{attribute 'qualified_only'}
{attribute 'strict'}
{attribute 'to_string'}
TYPE eTcaStorageCmd :
(
	noCmd := 0,
	FillCarrier,
	RemoveCarrier,
	EmptyCarrier
);
END_TYPE

(* stored: Version 1.1.0.1
   DUT eTcaStorageCmd: Id {d4b4f0ca-750b-4159-a9c0-0df2992c88b5} *)
